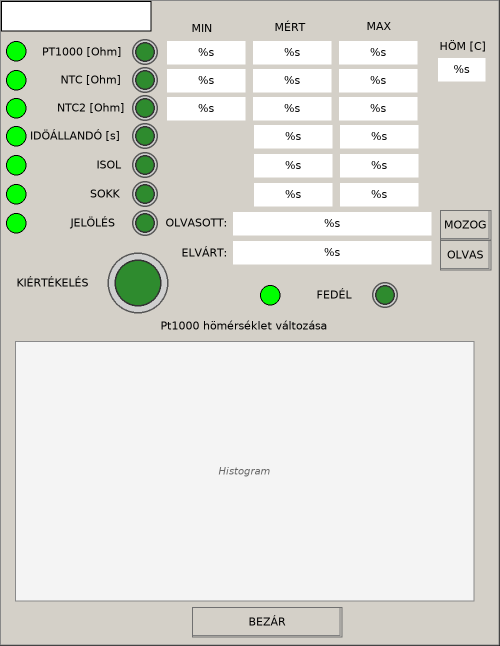
VISUALIZATION Meresek  // 500x646
    Rectangle (0,0 500x646)
    Lamp1 (130,150 30x30), variable: NOT GVL.bIsolOK, style: Lamp-Lamp1-Red
    Label (92,155 34x20), "ISOL"
    Label (182,16 40x25), "MIN"
    Histogram (15,341 459x260), scale format: %.1f, scale 0..300
        p1518820177: VEGMERO.arIdoallandoPTTEMP
        p102497268: VEGMERO.arIdoallandoPTTEMP
        p788070771: ARRAY [0..600] OF REAL
    Lamp1 (130,179 30x30), variable: NOT GVL.bShockOK, style: Lamp-Lamp1-Red
    Label (84,184 42x20), "SOKK"
    Label (60,213 66x20), "JELÖLÉS"
    Lamp1 (130,208 30x30), variable: NOT GVL.bMarkingOK, style: Lamp-Lamp1-Red
    Lamp1 (103,248 70x70), variable: GVL.bProductNOK, style: Lamp-Lamp1-Red
    Lamp1 (103,248 70x70), variable: GVL.bProductOK, invisible if: GVL.bProductNOK, style: Lamp-Lamp1-Green
    Label (7,268 91x30), "KIÉRTÉKELÉS"
    Label (38,42 88x20), "PT1000 [Ohm]"
    Lamp1 (130,37 30x30), variable: NOT GVL.bPTResOK, style: Lamp-Lamp1-Red
    Textfield (252,40 80x25), "%s", text variable: GVL.rPtRes
    Textfield (166,40 80x25), "%s", text variable: VEGMERO.PTRES_MIN
    Textfield (338,40 80x25), "%s", text variable: VEGMERO.PTRES_MAX
    Label (56,70 70x20), "NTC [Ohm]"
    Lamp1 (130,65 30x30), variable: NOT GVL.bNTCResOK, style: Lamp-Lamp1-Red
    Textfield (252,68 80x25), "%s", text variable: GVL.rNTCRes
    Textfield (166,68 80x25), "%s", text variable: VEGMERO.NTCRES_MIN
    Textfield (338,68 80x25), "%s", text variable: VEGMERO.NTCRES_MAX
    Lamp1 (130,121 30x30), variable: NOT GVL.bTimeConstOK, style: Lamp-Lamp1-Red
    Label (24,126 102x20), "IDÖÁLLANDÓ [s]"
    Textfield (253,124 80x25), "%s", text variable: GVL.rTimeConst
    Textfield (437,57 49x25), "%s", text variable: GVL.rTemp
    Label (359,14 40x25), "MAX"
    Label (270,15 40x25), "MÉRT"
    Label (438,34 50x25), "HÖM [C]"
    Textfield (339,124 80x25), "%s", text variable: REAL_TO_TIME(GVL.rIdoallandoMax*1000)
    Label (144,311 200x30), "Pt1000 hömérséklet változása"
    Textfield (253,153 80x25), "%s", text variable: VEGMERO.rISOL
    Textfield (339,153 80x25), "%s", text variable: GVL.rISOL_MAX
    Textfield (232,211 200x25), "%s", text variable: ZEBRASCANNER.sReceivedString255
    Button (192,607 150x30), "BEZÁR", invisible if: GVL.bMeresiEredmenyekRejtve
        OnMouseUp: execute { GVL.bMeresiEredmenyekRejtve:=TRUE; }
    Textfield (232,240 200x25), "%s", text variable: AUTOMATA.sExpectedCode
    Label (164,213 66x20), "OLVASOTT:"
    Label (164,243 66x20), "ELVÁRT:"
    Textfield (253,182 80x25), "%s", text variable: GVL.rPtResShock
    Textfield (339,182 80x25), "%s", text variable: GVL.PTRES_SOKK_MAX
    Lamp1 (130,37 30x30), variable: GVL.bPTResOK, invisible if: NOT GVL.bPTResOK AND VEGMERO.bPTRES_MERVE, style: Lamp-Lamp1-Green
    Lamp1 (130,150 30x30), variable: GVL.bIsolOK, invisible if: NOT GVL.bIsolOK AND VEGMERO.bISOL_MERVE, style: Lamp-Lamp1-Green
    Lamp1 (130,179 30x30), variable: GVL.bShockOK, invisible if: NOT GVL.bShockOK AND VEGMERO.bSOKK_MERVE, style: Lamp-Lamp1-Green
    Lamp1 (130,208 30x30), variable: GVL.bMarkingOK, invisible if: NOT GVL.bMarkingOK AND GVL.bMarking_ellenorizve, style: Lamp-Lamp1-Green
    Lamp1 (130,65 30x30), variable: GVL.bNTCResOK, invisible if: NOT GVL.bNTCResOK AND VEGMERO.bNTCRES_MERVE, style: Lamp-Lamp1-Green
    Lamp1 (130,121 30x30), variable: GVL.bTimeConstOK, invisible if: NOT GVL.bTimeConstOK AND VEGMERO.bIDOALLANDO_MERVE, style: Lamp-Lamp1-Green
    Ellipse (6,41 20x20), colour toggle: AUTOMATA.iProductTypeUnderTest<-1, invisible if: NOT GVL.bMeresBe
    Ellipse (6,70 20x20), colour toggle: AUTOMATA.iProductTypeUnderTest<-1, invisible if: NOT GVL.bMeresBe
    Ellipse (6,126 20x20), invisible if: (AUTOMATA.iProductTypeUnderTest<-1) OR NOT GVL.bMeresBe
    Ellipse (6,155 20x20), colour toggle: AUTOMATA.iProductTypeUnderTest=-2, invisible if: NOT GVL.bMeresBe
    Ellipse (6,213 20x20), invisible if: NOT GVL.bMeresBe
    Ellipse (6,184 20x20), invisible if: (AUTOMATA.iProductTypeUnderTest<0) OR NOT GVL.bMeresBe
    Label (290,285 88x20), "FEDÉL"
    Lamp1 (370,280 30x30), variable: GVL.bFedelOK OR GVL.bHimbaOK, style: Lamp-Lamp1-Green
    Ellipse (260,285 20x20), colour toggle: AUTOMATA.iProductTypeUnderTest<-2, invisible if: NOT GVL.bMeresBe
    Rectangle (1,1 150x30), text list: 'DUT_types', text index: GVL.iCurrentProductType+3
    Ellipse (6,98 20x20), colour toggle: AUTOMATA.iProductTypeUnderTest<-1, invisible if: NOT GVL.bMeresBe OR (GVL.iSelectedProductType<8)
    Label (56,98 70x20), "NTC2 [Ohm]"
    Textfield (252,96 80x25), "%s", text variable: GVL.rNTCRes2
    Textfield (166,96 80x25), "%s", text variable: VEGMERO.NTCRES2_MIN
    Textfield (338,96 80x25), "%s", text variable: VEGMERO.NTCRES2_MAX
    Lamp1 (130,93 30x30), variable: NOT GVL.bNTCRes2OK, style: Lamp-Lamp1-Red
    Lamp1 (130,93 30x30), variable: GVL.bNTCRes2OK, invisible if: NOT GVL.bNTCRes2OK AND VEGMERO.bNTCRES2_MERVE, style: Lamp-Lamp1-Green
    Button (440,210 51x30), "MOZOG"
        OnMouseUp: execute { PISTITENGELY.lrPistiPosition:=GVL.lrKodolvasasPosition; PISTITENGELY.sPistiAxisCommand:='MOVE'; }
    Button (440,240 51x30), "OLVAS"
        OnMouseUp: execute { ZEBRASCANNER.bStartSend:=true; }
END_VISUALIZATION

(* stored: Version 1.1.0.1, ProductVersion 3.1.4024.11
   Visu Meresek: Id {b5e0f60c-96ae-4843-baef-a1a008f5081d} *)
